// TIA Portal V17 export
// export: Created 2024-08-09T12:50:43.4109306Z, ExportSetting WithDefaults, DisplayName Totally Integrated Automation Portal, DisplayVersion V17 Update 7, DisplayName TIA Portal Openness, DisplayVersion V17 Update 7, DisplayName TIA Portal Version Control Interface, DisplayVersion V17, DisplayName STEP 7 Professional, DisplayVersion V17 Update 7, DisplayName STEP 7 Safety, DisplayVersion V17 Update 6, DisplayName WinCC Professional, DisplayVersion V17 Update 7
DATA_BLOCK "fbSql4SiemensConnectionObserver3_DB"   // DB29
VERSION : 0.1
// stored: AutoNumber true, DBAccessibleFromOPCUA true, DBAccessibleFromWebserver true, InstanceOfName fbSql4SiemensConnectionObserver3, InstanceOfType FB
"fbSql4SiemensConnectionObserver3"
   // VAR_INPUT
   //    tTimeout : Time;
   //    xCloseConnection : Bool;
   // END_VAR
   // VAR_IN_OUT
   //    stSql4SiemensInterface : "utSql4SiemensInterface";
   // END_VAR
   // VAR
   //    inTimeout { S7_SetPoint := 'True'} : TON_TIME;
   //    iStep : Int;
   //    diDoneCount : DInt;
   //    diErrorCount : DInt;
   // END_VAR
BEGIN
END_DATA_BLOCK
